{attribute 'qualified_only'}
VAR_GLOBAL
	
	stMotors		: ST_Motors;
	
	// coolingMotor		: FB_MotorFq
END_VAR

(* stored: Version 1.1.0.1
   GVL Motors: Id {0fd1bec4-5ad5-43cb-9c61-d003cd78f966} *)
